TYPE T_ALIAS : WORD;
END_TYPE

(* stored: Version 1.1.0.1, ProductVersion 3.1.4024.11
   DUT T_ALIAS: Id {211c8563-7ef4-49a4-abc1-63eb79b1eac8} *)
